// TIA Portal V17 export
// export: Created 2025-03-07T09:24:00.8247704Z, ExportSetting WithDefaults, DisplayName Totally Integrated Automation Portal, DisplayVersion V17 Update 8, DisplayName TIA Portal Openness, DisplayVersion V17 Update 8, DisplayName TIA Portal Version Control Interface, DisplayVersion V17, DisplayName SINAMICS Startdrive Advanced, DisplayVersion V17 SP2, DisplayName SINAMICS Startdrive G110M, G120, G120C, G120D, G120P, G115D, DisplayVersion V17 SP2, DisplayName SINAMICS Startdrive G130, G150, S120, S150, SINAMICS MV, S210, DisplayVersion V17 SP2, DisplayName STEP 7 Professional, DisplayVersion V17 Update 8, DisplayName SINUMERIK ONE STEP 7 Toolbox, DisplayVersion V17 Update 12, DisplayName SINUMERIK 840D sl STEP 7 Toolbox, DisplayVersion V17 Update 12, DisplayName STEP 7 Safety, DisplayVersion V17 Update 6, DisplayName WinCC Advanced, DisplayVersion V17 Update 8
DATA_BLOCK "DB21025_POWDER_FEEDER_1_PROFINET_UNIT_02"   // DB21025
{ DB_Accessible_From_OPC_UA := 'FALSE' }
VERSION : 0.1
// stored: AutoNumber false, DBAccessibleFromOPCUA false, DBAccessibleFromWebserver true, InstanceOfName FB21014_POWDER_FEEDER_PROFINET, InstanceOfType FB
"FB21014_POWDER_FEEDER_PROFINET"
   // VAR_INPUT
   //    "iHMI_Values Setpoints" : "POWDER FEEDER HMI VALUES SETPOINTS";
   //    "iHMI_Offsets Alarms and Warnings" : "POWDER FEEDER HMI OFFSETS ALARMS WARNINGS";
   //    "iCNC_Values Setpoints" : "POWDER FEEDER CNC VALUES SETPOINTS";
   //    iSTOP_LINE_1_VALUES_SETPOINTS : Struct
   //       LINE_1_GAS_FLOW : Real;
   //       LINE_1_DISK_SPEED : Real;
   //    END_STRUCT;
   //    iSTOP_LINE_2_VALUES_SETPOINTS : Struct
   //       LINE_2_GAS_FLOW : Real;
   //       LINE_2_DISK_SPEED : Real;
   //    END_STRUCT;
   //    iSTART_LINE_1_VALUES_SETPOINTS : Struct
   //       LINE_1_GAS_FLOW : Real;
   //       LINE_1_DISK_SPEED : Real;
   //    END_STRUCT;
   //    iSTART_LINE_2_VALUES_SETPOINTS : Struct
   //       LINE_2_GAS_FLOW : Real;
   //       LINE_2_DISK_SPEED : Real;
   //    END_STRUCT;
   //    iArgon_Carrier_Gas_Selected : Bool;
   //    iNitro_Carrier_Gas_Selected : Bool;
   //    iHelium_Carrier_Gas_Selected : Bool;
   //    iArgon30_Carrier_Gas_Selected : Bool;
   //    iLINE_1_ON_SEQ_ON : Bool;
   //    iLINE_2_ON_SEQ_ON : Bool;
   //    iLINE_1_OFF_SEQ_ON : Bool;
   //    iLINE_2_OFF_SEQ_ON : Bool;
   //    iLINE_1_STOPPED : Bool;
   //    iLINE_2_STOPPED : Bool;
   // END_VAR
   // VAR_OUTPUT
   //    oPLC_Aux : "POWDER FEEDER PLC AUXILIAR";
   //    oSTATION_WARNINGS : Bool;
   //    oWARNING_PF_LINE_1_GRAVIMETRIC_MODE_SELECTED : Bool;
   //    oWARNING_PF_LINE_2_GRAVIMETRIC_MODE_SELECTED : Bool;
   // END_VAR
   // VAR_IN_OUT
   //    ioPowder_Feeder_Unit_In_Out : "POWDER FEEDER OERLIKON";
   // END_VAR
   // VAR RETAIN
   //    INPUT_SETTINGS : Struct
   //       UNIT_NUMBER : Int;
   //       FEEDER_NUMBER : Int;
   //    END_STRUCT;
   //    AUX_MANUAL_GAS_LINE_1 : Bool;
   //    AUX_MANUAL_GAS_LINE_2 : Bool;
   //    AUX_MANUAL_DISK_LINE_1 : Bool;
   //    AUX_MANUAL_DISK_LINE_2 : Bool;
   //    swapped : Word;
   // END_VAR
BEGIN
END_DATA_BLOCK
